TYPE ST_PTOStepperRef :
STRUCT
	nCounterValue 		AT %I* : UINT;
	bCounterUnderflow	AT %I* : BOOL;
	bCounterOverflow	AT %I* : BOOL;
	bSetCounter			AT %Q* : BOOL;
	nFrequencyValue 	AT %Q* : UINT;
	nSetCounterValue	AT %Q* : UINT;
END_STRUCT
END_TYPE

(* stored: Version 1.1.0.1, ProductVersion 3.1.4020.12
   DUT ST_PTOStepperRef: Id {98ef2670-4f1e-4d4c-89f0-d5ebf8de3599} *)
